{attribute 'qualified_only'}
{attribute 'strict'}
TYPE E_MbXferState :
(
	Idle := 0,
	Busy,
	Done,
	Timeout,
	Error
);
END_TYPE

(* stored: Version 1.1.0.1
   DUT E_MbXferState: Id {a26a28f5-ef32-41b7-93e2-193455efa28d} *)
